// TIA Portal V16 export
// export: Created 2021-09-08T12:46:12.3893396Z, ExportSetting WithDefaults, DisplayName Totally Integrated Automation Portal, DisplayVersion V16 Update 3, DisplayName TIA Portal Version Control Interface, DisplayVersion V16 Update 2, DisplayName TIA Portal Openness, DisplayVersion V16 Update 3, DisplayName TIA Portal Teamcenter Gateway, DisplayVersion V16, DisplayName STEP 7 Professional, DisplayVersion V16 Update 3, DisplayName STEP 7 Safety, DisplayVersion V16, DisplayName WinCC Advanced, DisplayVersion V16 Update 3
FUNCTION_BLOCK "AllDigital"   // FB5, FBD
{ S7_Optimized_Access := 'TRUE' }
VERSION : 0.1
// stored: AutoNumber true, IsIECCheckEnabled false, IsRetainMemResEnabled false, MemoryReserve 100, SetENOAutomatically false, UDAEnableTagReadback false
   VAR
      FL501 { S7_SetPoint := 'True'} : "DigitalSensorCntrl";
      FL901 { S7_SetPoint := 'True'} : "DigitalSensorCntrl";
      FL1301 { S7_SetPoint := 'True'} : "DigitalSensorCntrl";
      PS901 { S7_SetPoint := 'True'} : "DigitalSensorCntrl";
      PS902 { S7_SetPoint := 'True'} : "DigitalSensorCntrl";
      PS1301 { S7_SetPoint := 'True'} : "DigitalSensorCntrl";
      PS1302 { S7_SetPoint := 'True'} : "DigitalSensorCntrl";
   END_VAR
BEGIN

REGION Network 1: 1-включить детектирование аварии
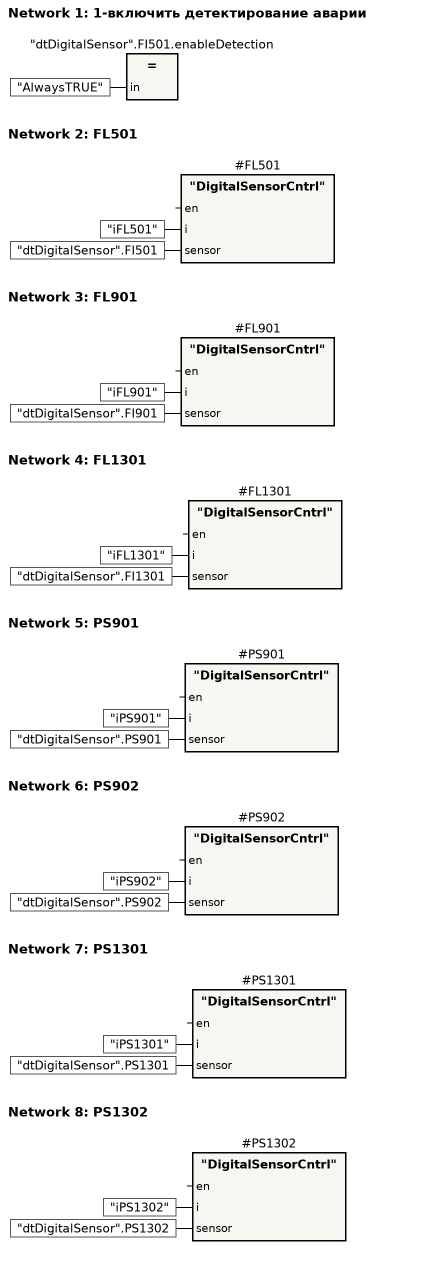
   "dtDigitalSensor".FI501.enableDetection := "AlwaysTRUE";
END_REGION

REGION Network 2: FL501
   #FL501(i := "iFL501", sensor := "dtDigitalSensor".FI501);   // "DigitalSensorCntrl"
END_REGION

REGION Network 3: FL901
   #FL901(i := "iFL901", sensor := "dtDigitalSensor".FI901);   // "DigitalSensorCntrl"
END_REGION

REGION Network 4: FL1301
   #FL1301(i := "iFL1301", sensor := "dtDigitalSensor".FI1301);   // "DigitalSensorCntrl"
END_REGION

REGION Network 5: PS901
   #PS901(i := "iPS901", sensor := "dtDigitalSensor".PS901);   // "DigitalSensorCntrl"
END_REGION

REGION Network 6: PS902
   #PS902(i := "iPS902", sensor := "dtDigitalSensor".PS902);   // "DigitalSensorCntrl"
END_REGION

REGION Network 7: PS1301
   #PS1301(i := "iPS1301", sensor := "dtDigitalSensor".PS1301);   // "DigitalSensorCntrl"
END_REGION

REGION Network 8: PS1302
   #PS1302(i := "iPS1302", sensor := "dtDigitalSensor".PS1302);   // "DigitalSensorCntrl"
END_REGION
END_FUNCTION_BLOCK
